ABB RAPID module: MAINMODULE

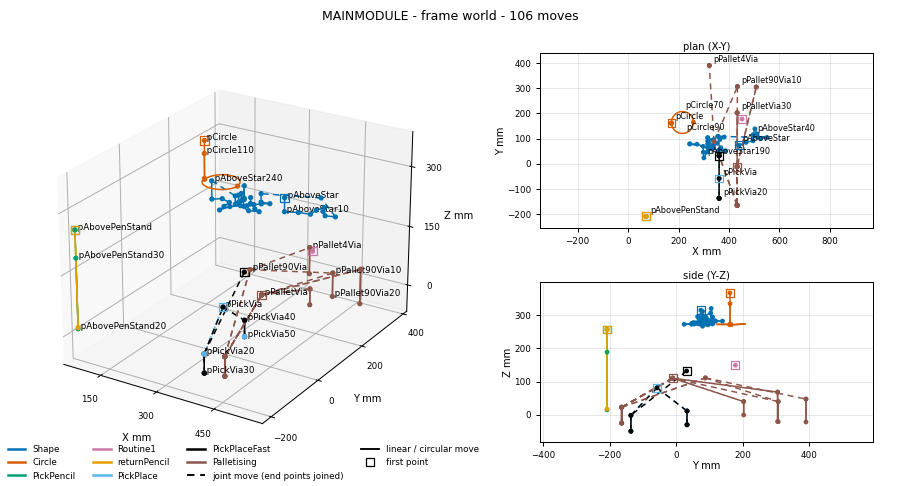
[picture p0: tool path of MAINMODULE in frame world, 106 of 141 moves have a stored position in this frame; points joined in program order, loops and branches not executed]
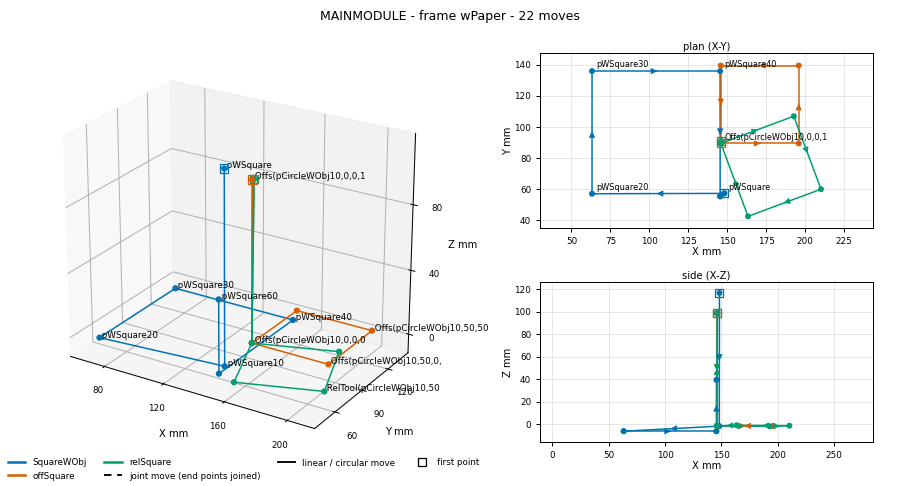
[picture p1: tool path of MAINMODULE in frame wPaper, 22 of 141 moves have a stored position in this frame; points joined in program order, loops and branches not executed]
MODULE MainModule
	CONST robtarget pAboveStar:=[[438.62,74.11,314.72],[0.00782336,-0.999705,-0.0203543,-0.0106794],[0,0,2,0],[9E+09,9E+09,9E+09,9E+09,9E+09,9E+09]];
	CONST robtarget pAboveStar10:=[[438.61,74.11,281.38],[0.00783533,-0.999705,-0.0203361,-0.0106734],[0,0,2,0],[9E+09,9E+09,9E+09,9E+09,9E+09,9E+09]];
	CONST robtarget pAboveStar20:=[[467.60,85.46,281.94],[0.00786178,-0.999706,-0.0202732,-0.0107677],[0,0,2,0],[9E+09,9E+09,9E+09,9E+09,9E+09,9E+09]];
	CONST robtarget pAboveStar30:=[[494.86,91.66,281.75],[0.00785369,-0.999704,-0.0202728,-0.010905],[0,0,2,0],[9E+09,9E+09,9E+09,9E+09,9E+09,9E+09]];
	CONST robtarget pAboveStar40:=[[495.39,115.61,282.55],[0.00784958,-0.999705,-0.0202499,-0.0109168],[0,0,2,0],[9E+09,9E+09,9E+09,9E+09,9E+09,9E+09]];
	CONST robtarget pAboveStar50:=[[502.60,139.11,282.02],[0.00780388,-0.999706,-0.0202427,-0.0108406],[0,0,2,0],[9E+09,9E+09,9E+09,9E+09,9E+09,9E+09]];
	CONST robtarget pAboveStar60:=[[511.39,118.70,282.17],[0.00782157,-0.999704,-0.0203071,-0.010834],[0,0,2,0],[9E+09,9E+09,9E+09,9E+09,9E+09,9E+09]];
	CONST robtarget pAboveStar70:=[[526.59,101.47,281.57],[0.00783068,-0.999704,-0.0203263,-0.0108239],[0,0,2,0],[9E+09,9E+09,9E+09,9E+09,9E+09,9E+09]];
	CONST robtarget pAboveStar80:=[[550.47,105.19,283.01],[0.00780734,-0.999704,-0.020355,-0.0107971],[0,0,2,0],[9E+09,9E+09,9E+09,9E+09,9E+09,9E+09]];
	CONST robtarget pAboveStar90:=[[513.27,105.19,320.11],[0.00778152,-0.999706,-0.0203135,-0.010705],[0,0,2,0],[9E+09,9E+09,9E+09,9E+09,9E+09,9E+09]];
	CONST robtarget pAboveStar100:=[[356.24,109.54,273.41],[0.0140382,0.0113166,0.999798,0.00891365],[0,0,0,0],[9E+09,9E+09,9E+09,9E+09,9E+09,9E+09]];
	CONST robtarget pAboveStar110:=[[381.12,106.70,276.14],[0.0141146,0.0112878,0.999797,0.00891807],[0,0,0,0],[9E+09,9E+09,9E+09,9E+09,9E+09,9E+09]];
	CONST robtarget pAboveStar120:=[[364.27,97.27,275.21],[0.0140659,0.0112485,0.999798,0.00892909],[0,0,0,0],[9E+09,9E+09,9E+09,9E+09,9E+09,9E+09]];
	CONST robtarget pAboveStar130:=[[353.90,82.53,276.31],[0.0142624,0.0112492,0.999794,0.00900628],[0,0,0,0],[9E+09,9E+09,9E+09,9E+09,9E+09,9E+09]];
	CONST robtarget pAboveStar140:=[[367.61,64.33,275.67],[0.0143661,0.0112371,0.999793,0.00904389],[0,0,0,0],[9E+09,9E+09,9E+09,9E+09,9E+09,9E+09]];
	CONST robtarget pAboveStar150:=[[386.45,52.10,277.62],[0.0144419,0.0112929,0.999791,0.00908413],[0,0,0,0],[9E+09,9E+09,9E+09,9E+09,9E+09,9E+09]];
	CONST robtarget pAboveStar160:=[[358.13,53.57,273.11],[0.0145648,0.011269,0.999789,0.00914371],[0,0,0,0],[9E+09,9E+09,9E+09,9E+09,9E+09,9E+09]];
	CONST robtarget pAboveStar170:=[[332.66,60.20,277.10],[0.0146625,0.0112876,0.999787,0.00917015],[0,0,0,0],[9E+09,9E+09,9E+09,9E+09,9E+09,9E+09]];
	CONST robtarget pAboveStar180:=[[313.01,46.92,275.35],[0.0146979,0.011265,0.999786,0.00921032],[0,0,0,0],[9E+09,9E+09,9E+09,9E+09,9E+09,9E+09]];
	CONST robtarget pAboveStar190:=[[300.34,23.93,272.39],[0.0147404,0.0112439,0.999785,0.00926598],[0,0,0,0],[9E+09,9E+09,9E+09,9E+09,9E+09,9E+09]];
	CONST robtarget pAboveStar200:=[[297.97,46.30,272.71],[0.0147271,0.0111926,0.999785,0.00933937],[0,0,0,0],[9E+09,9E+09,9E+09,9E+09,9E+09,9E+09]];
	CONST robtarget pAboveStar210:=[[297.39,69.49,273.85],[0.0147374,0.0111578,0.999785,0.00935574],[0,0,0,0],[9E+09,9E+09,9E+09,9E+09,9E+09,9E+09]];
	CONST robtarget pAboveStar220:=[[272.94,78.27,274.40],[0.0147777,0.0111411,0.999784,0.00940734],[0,0,0,0],[9E+09,9E+09,9E+09,9E+09,9E+09,9E+09]];
	CONST robtarget pAboveStar230:=[[244.38,79.32,266.59],[0.0148682,0.0111358,0.999783,0.00945356],[0,0,0,0],[9E+09,9E+09,9E+09,9E+09,9E+09,9E+09]];
	CONST robtarget pAboveStar240:=[[244.38,79.32,311.23],[0.0148422,0.0111395,0.999783,0.00942161],[0,0,0,0],[9E+09,9E+09,9E+09,9E+09,9E+09,9E+09]];
	CONST robtarget pAboveStar250:=[[356.24,109.54,293.90],[0.014005,0.0113197,0.999798,0.00888656],[0,0,0,0],[9E+09,9E+09,9E+09,9E+09,9E+09,9E+09]];
	CONST robtarget pAboveStar260:=[[316.18,64.48,295.54],[0.0148764,0.0111011,0.999783,0.00946381],[0,0,0,0],[9E+09,9E+09,9E+09,9E+09,9E+09,9E+09]];
	CONST robtarget pAboveStar270:=[[316.19,64.48,275.26],[0.0149083,0.0111043,0.999782,0.00947887],[0,0,0,0],[9E+09,9E+09,9E+09,9E+09,9E+09,9E+09]];
	CONST robtarget pAboveStar280:=[[319.92,71.32,275.46],[0.0149256,0.0110552,0.999782,0.00950374],[0,0,0,0],[9E+09,9E+09,9E+09,9E+09,9E+09,9E+09]];
	CONST robtarget pAboveStar290:=[[316.12,78.28,275.06],[0.0149297,0.0109983,0.999783,0.00948498],[0,0,0,0],[9E+09,9E+09,9E+09,9E+09,9E+09,9E+09]];
	CONST robtarget pAboveStar300:=[[316.12,78.28,292.53],[0.0149053,0.0110043,0.999784,0.00945692],[0,0,0,0],[9E+09,9E+09,9E+09,9E+09,9E+09,9E+09]];
	CONST robtarget pAboveStar310:=[[316.11,90.07,292.53],[0.0148157,0.0109983,0.999785,0.00941225],[0,0,0,0],[9E+09,9E+09,9E+09,9E+09,9E+09,9E+09]];
	CONST robtarget pAboveStar320:=[[316.13,90.08,275.06],[0.0150005,0.0109958,0.999782,0.00946723],[0,0,0,0],[9E+09,9E+09,9E+09,9E+09,9E+09,9E+09]];
	CONST robtarget pAboveStar330:=[[319.37,97.08,275.77],[0.015104,0.0109807,0.999781,0.009478],[0,0,0,0],[9E+09,9E+09,9E+09,9E+09,9E+09,9E+09]];
	CONST robtarget pAboveStar340:=[[315.40,103.87,275.53],[0.0151335,0.0110028,0.99978,0.00947056],[0,0,0,0],[9E+09,9E+09,9E+09,9E+09,9E+09,9E+09]];
	CONST robtarget pAboveStar350:=[[315.40,103.86,306.27],[0.0151151,0.0109962,0.999781,0.00943505],[0,0,0,0],[9E+09,9E+09,9E+09,9E+09,9E+09,9E+09]];
	CONST robtarget pAboveStar360:=[[335.06,68.19,290.35],[0.015148,0.0110168,0.99978,0.00946204],[0,0,0,0],[9E+09,9E+09,9E+09,9E+09,9E+09,9E+09]];
	CONST robtarget pAboveStar370:=[[336.39,68.12,273.72],[0.0152631,0.0109898,0.999778,0.0095098],[0,0,0,0],[9E+09,9E+09,9E+09,9E+09,9E+09,9E+09]];
	CONST robtarget pAboveStar380:=[[339.60,77.00,272.41],[0.0152849,0.0109759,0.999778,0.00952187],[0,0,0,0],[9E+09,9E+09,9E+09,9E+09,9E+09,9E+09]];
	CONST robtarget pAboveStar390:=[[341.03,87.53,273.01],[0.0152756,0.0109779,0.999778,0.0095199],[0,0,0,0],[9E+09,9E+09,9E+09,9E+09,9E+09,9E+09]];
	CONST robtarget pAboveStar400:=[[337.71,95.21,270.79],[0.015379,0.0110505,0.999775,0.00953919],[0,0,0,0],[9E+09,9E+09,9E+09,9E+09,9E+09,9E+09]];
	CONST robtarget pAboveStar410:=[[337.71,95.21,285.45],[0.0153497,0.0110536,0.999776,0.00950113],[0,0,0,0],[9E+09,9E+09,9E+09,9E+09,9E+09,9E+09]];
	CONST robtarget pCircle:=[[172.19,161.39,366.69],[0.0151956,0.0110729,0.999778,0.00948806],[0,-1,0,0],[9E+09,9E+09,9E+09,9E+09,9E+09,9E+09]];
	CONST robtarget pCircle10:=[[172.21,161.39,272.61],[0.0153553,0.0110984,0.999775,0.00956675],[0,-1,0,0],[9E+09,9E+09,9E+09,9E+09,9E+09,9E+09]];
	CONST robtarget pCircle30:=[[172.21,161.40,271.86],[0.0153361,0.0111049,0.999775,0.00957292],[0,-1,0,0],[9E+09,9E+09,9E+09,9E+09,9E+09,9E+09]];
	CONST robtarget pCircle20:=[[172.21,161.40,271.86],[0.0153361,0.0111049,0.999775,0.00957292],[0,-1,0,0],[9E+09,9E+09,9E+09,9E+09,9E+09,9E+09]];
	CONST robtarget pCircle40:=[[172.20,161.39,270.86],[0.0153246,0.0111176,0.999775,0.00958173],[0,-1,0,0],[9E+09,9E+09,9E+09,9E+09,9E+09,9E+09]];
	CONST robtarget pCircle60:=[[172.20,161.39,271.86],[0.0153102,0.0111183,0.999775,0.00956012],[0,-1,0,0],[9E+09,9E+09,9E+09,9E+09,9E+09,9E+09]];
	CONST robtarget pCircle50:=[[172.20,161.39,271.86],[0.0153102,0.0111183,0.999775,0.00956012],[0,-1,0,0],[9E+09,9E+09,9E+09,9E+09,9E+09,9E+09]];
	CONST robtarget pCircle80:=[[258.72,165.57,271.21],[0.0155733,0.0111395,0.999769,0.00972795],[0,-1,0,0],[9E+09,9E+09,9E+09,9E+09,9E+09,9E+09]];
	CONST robtarget pCircle70:=[[213.26,207.69,273.19],[0.0153849,0.0111178,0.999772,0.00975547],[0,-1,0,0],[9E+09,9E+09,9E+09,9E+09,9E+09,9E+09]];
	CONST robtarget pCircle100:=[[171.43,161.80,272.76],[0.0157088,0.0111,0.999768,0.00974234],[0,-1,0,0],[9E+09,9E+09,9E+09,9E+09,9E+09,9E+09]];
	CONST robtarget pCircle90:=[[217.30,120.93,272.13],[0.0155276,0.0111561,0.99977,0.00968626],[0,0,0,0],[9E+09,9E+09,9E+09,9E+09,9E+09,9E+09]];
	CONST robtarget pCircle110:=[[171.42,161.80,334.48],[0.0156731,0.0110978,0.999768,0.00974344],[0,-1,0,0],[9E+09,9E+09,9E+09,9E+09,9E+09,9E+09]];
	CONST robtarget pPen:=[[164.19,-206.82,447.81],[0.0140855,0.999796,-0.00773344,0.0122549],[-1,0,1,0],[9E+09,9E+09,9E+09,9E+09,9E+09,9E+09]];
	CONST robtarget pPen10:=[[164.19,-206.82,255.83],[0.014113,0.999795,-0.00772477,0.0122876],[-1,0,1,0],[9E+09,9E+09,9E+09,9E+09,9E+09,9E+09]];
	CONST robtarget pPen20:=[[164.19,-206.82,402.79],[0.0141017,0.999795,-0.00773661,0.0122669],[-1,0,1,0],[9E+09,9E+09,9E+09,9E+09,9E+09,9E+09]];
	CONST robtarget pWSquare:=[[148.16,57.39,116.56],[0.00760039,0.985996,-0.166519,0.00508158],[0,0,0,0],[9E+09,9E+09,9E+09,9E+09,9E+09,9E+09]];
	CONST robtarget pWSquare10:=[[148.04,57.38,-1.61],[0.00765696,0.985998,-0.166511,0.00489645],[0,0,0,0],[9E+09,9E+09,9E+09,9E+09,9E+09,9E+09]];
	CONST robtarget pWSquare20:=[[63.18,57.15,-6.08],[0.00767438,0.986016,-0.166404,0.00479981],[0,0,0,0],[9E+09,9E+09,9E+09,9E+09,9E+09,9E+09]];
	CONST robtarget pWSquare30:=[[63.20,135.93,-6.09],[0.00763878,0.986022,-0.166368,0.00484462],[0,0,0,0],[9E+09,9E+09,9E+09,9E+09,9E+09,9E+09]];
	CONST robtarget pWSquare40:=[[145.43,135.93,-6.09],[0.00764315,0.986027,-0.166343,0.00481764],[0,0,0,0],[9E+09,9E+09,9E+09,9E+09,9E+09,9E+09]];
	CONST robtarget pWSquare50:=[[145.46,55.49,-6.09],[0.00763597,0.986023,-0.166361,0.00488827],[0,0,0,0],[9E+09,9E+09,9E+09,9E+09,9E+09,9E+09]];
	CONST robtarget pWSquare60:=[[145.48,55.51,39.46],[0.00758059,0.986027,-0.16634,0.00490909],[0,0,0,0],[9E+09,9E+09,9E+09,9E+09,9E+09,9E+09]];
	CONST robtarget pAbovePenStand:=[[71.07,-207.77,256.82],[0.00907654,-0.0280649,0.999549,0.00556097],[-2,-1,-2,0],[9E+09,9E+09,9E+09,9E+09,9E+09,9E+09]];
	CONST robtarget pAbovePenStand10:=[[71.05,-207.81,17.76],[0.00903694,-0.0280484,0.999551,0.00548002],[-2,-1,-2,0],[9E+09,9E+09,9E+09,9E+09,9E+09,9E+09]];
	CONST robtarget pAbovePenStand20:=[[71.05,-207.84,14.94],[0.00903621,-0.0280371,0.999551,0.00543696],[-2,-1,-2,0],[9E+09,9E+09,9E+09,9E+09,9E+09,9E+09]];
	CONST robtarget pAbovePenStand30:=[[71.07,-207.82,188.80],[0.00907619,-0.0280604,0.99955,0.00546786],[-2,-1,-2,0],[9E+09,9E+09,9E+09,9E+09,9E+09,9E+09]];
	CONST robtarget pCircleWObj:=[[145.95,89.49,175.26],[0.00623942,0.984129,0.177325,-0.0027726],[-1,-1,-1,0],[9E+09,9E+09,9E+09,9E+09,9E+09,9E+09]];
	CONST robtarget pCircleWObj10:=[[145.91,89.49,-1.38],[0.00623623,0.984131,0.17731,-0.0028463],[-1,-1,-1,0],[9E+09,9E+09,9E+09,9E+09,9E+09,9E+09]];
	CONST robtarget pCircleWObj30:=[[59.69,88.08,-0.69],[0.00626669,0.984148,0.177212,-0.00309014],[-1,-1,-1,0],[9E+09,9E+09,9E+09,9E+09,9E+09,9E+09]];
	CONST robtarget pCircleWObj20:=[[104.28,44.81,0.78],[0.00625793,0.984143,0.17724,-0.00298966],[-1,-1,-1,0],[9E+09,9E+09,9E+09,9E+09,9E+09,9E+09]];
	CONST robtarget pCircleWObj50:=[[146.50,89.95,0.21],[0.00622075,0.984144,0.177231,-0.00332268],[-1,-1,-1,0],[9E+09,9E+09,9E+09,9E+09,9E+09,9E+09]];
	CONST robtarget pCircleWObj40:=[[102.61,131.54,-0.10],[0.00622868,0.984143,0.17724,-0.00320295],[-1,-1,-1,0],[9E+09,9E+09,9E+09,9E+09,9E+09,9E+09]];
	CONST robtarget pCircleWObj60:=[[146.53,89.93,120.78],[0.00626536,0.98414,0.17725,-0.00328061],[-1,-1,-1,0],[9E+09,9E+09,9E+09,9E+09,9E+09,9E+09]];
	CONST robtarget pTriangleWObj:=[[146.59,89.92,166.63],[0.00627944,0.984134,0.177285,-0.00319599],[-1,-1,-1,0],[9E+09,9E+09,9E+09,9E+09,9E+09,9E+09]];
	CONST robtarget pTriangleWObj10:=[[146.61,89.93,-1.46],[0.00627066,0.984138,0.177267,-0.00317229],[-1,-1,-1,0],[9E+09,9E+09,9E+09,9E+09,9E+09,9E+09]];
	CONST robtarget pTriangleWObj20:=[[72.70,56.70,-2.34],[0.00625777,0.984117,0.177377,-0.00333694],[-1,-1,-1,0],[9E+09,9E+09,9E+09,9E+09,9E+09,9E+09]];
	CONST robtarget pTriangleWObj30:=[[72.63,118.18,-0.40],[0.00623532,0.984124,0.177339,-0.00344523],[-1,-1,-1,0],[9E+09,9E+09,9E+09,9E+09,9E+09,9E+09]];
	CONST robtarget pTriangleWObj40:=[[146.62,89.92,123.42],[0.00628958,0.984135,0.17728,-0.00316079],[-1,-1,-1,0],[9E+09,9E+09,9E+09,9E+09,9E+09,9E+09]];
	CONST robtarget pPickVia:=[[360.73,-57.78,81.44],[0.00903673,-0.0280459,0.99955,0.00558822],[-1,-1,-1,0],[9E+09,9E+09,9E+09,9E+09,9E+09,9E+09]];
	CONST robtarget pPickVia10:=[[389.78,-126.91,12.64],[0.00911789,-0.0280836,0.999549,0.00553206],[-1,-1,-1,0],[9E+09,9E+09,9E+09,9E+09,9E+09,9E+09]];
	CONST robtarget pPickAbove10:=[[389.83,-126.95,-54.60],[0.00917495,-0.028089,0.999548,0.0054678],[-1,-1,-1,0],[9E+09,9E+09,9E+09,9E+09,9E+09,9E+09]];
	VAR clock cClock;
	VAR num nClock:=0;
	VAR string strClock:="";
	CONST robtarget pPickVia20:=[[360.72,-136.09,-1.19],[0.00903325,-0.0281173,0.999548,0.00555723],[-1,-1,-1,0],[9E+09,9E+09,9E+09,9E+09,9E+09,9E+09]];
	CONST robtarget pPickVia30:=[[360.77,-136.11,-48.89],[0.00910119,-0.0281037,0.999548,0.00552285],[-1,-1,-1,0],[9E+09,9E+09,9E+09,9E+09,9E+09,9E+09]];
	CONST robtarget pPickVia40:=[[360.83,32.61,11.70],[0.00906001,-0.0279562,0.999552,0.00563834],[0,0,0,0],[9E+09,9E+09,9E+09,9E+09,9E+09,9E+09]];
	CONST robtarget pPickVia50:=[[360.77,32.61,-29.56],[0.00898145,-0.0279684,0.999553,0.00563244],[0,0,0,0],[9E+09,9E+09,9E+09,9E+09,9E+09,9E+09]];
	CONST robtarget pPalletVia:=[[432.15,-10.57,110.48],[0.00897623,-0.0279392,0.999553,0.00565143],[-1,-1,-1,0],[9E+09,9E+09,9E+09,9E+09,9E+09,9E+09]];
	CONST robtarget pPalletVia10:=[[432.23,-163.79,23.13],[0.0089389,-0.0279646,0.999553,0.00565939],[-1,-1,-1,0],[9E+09,9E+09,9E+09,9E+09,9E+09,9E+09]];
	CONST robtarget pPalletVia20:=[[432.27,-163.81,-24.59],[0.00902617,-0.0279489,0.999553,0.00561107],[-1,-1,-1,0],[9E+09,9E+09,9E+09,9E+09,9E+09,9E+09]];
	CONST robtarget pPalletVia30:=[[432.16,202.87,40.09],[0.00885039,-0.0278895,0.999556,0.00567707],[0,0,0,0],[9E+09,9E+09,9E+09,9E+09,9E+09,9E+09]];
	CONST robtarget pPalletVia40:=[[432.15,202.88,-0.16],[0.00885213,-0.0278772,0.999556,0.00571044],[0,0,0,0],[9E+09,9E+09,9E+09,9E+09,9E+09,9E+09]];
	CONST robtarget pPallet90Via:=[[340.81,87.79,111.35],[0.00246793,-0.695514,0.7183,0.0172898],[-1,-1,-1,0],[9E+09,9E+09,9E+09,9E+09,9E+09,9E+09]];
	CONST robtarget pPallet90Via10:=[[433.23,306.73,40.16],[0.0024531,-0.695614,0.718204,0.0172648],[0,0,-1,0],[9E+09,9E+09,9E+09,9E+09,9E+09,9E+09]];
	CONST robtarget pPallet90Via20:=[[433.26,306.73,-20.32],[0.00247707,-0.6956,0.718218,0.0172488],[0,0,-1,0],[9E+09,9E+09,9E+09,9E+09,9E+09,9E+09]];
	CONST robtarget pPallet3Via:=[[507.97,304.84,68.59],[0.00881255,-0.0279233,0.999556,0.00560182],[0,0,0,0],[9E+09,9E+09,9E+09,9E+09,9E+09,9E+09]];
	CONST robtarget pPallet3Via10:=[[507.99,304.87,-19.58],[0.00883866,-0.0279657,0.999554,0.005633],[0,0,0,0],[9E+09,9E+09,9E+09,9E+09,9E+09,9E+09]];
	CONST robtarget pPallet4Via:=[[321.86,390.09,47.64],[0.00242,-0.695518,0.718297,0.0172813],[0,0,-1,0],[9E+09,9E+09,9E+09,9E+09,9E+09,9E+09]];
	CONST robtarget pPallet4Via10:=[[321.86,390.10,-21.25],[0.00243516,-0.695493,0.71832,0.0173165],[0,0,-1,0],[9E+09,9E+09,9E+09,9E+09,9E+09,9E+09]];
	PROC main()
		IF diSwitch1 = 1 AND diPenStand = 1 THEN
			PickPencil;
		ELSEIF diSwitch1 = 0 AND diPenStand = 0 THEN
			returnPencil;
		ENDIF
		IF diSwitch2 = 1 AND diGripSensor = 1 THEN
			nCircleNum := 0;
			FOR i FROM 1 TO 3 DO
				CircleWObj;
				Add nCircleNum, 1;
			ENDFOR
			UIMsgBox "3 circles drawn.";
		ELSEIF FALSE AND diGripSensor = 1 THEN
            nTriangleNum := 0;
			FOR i FROM 1 TO 3 DO
				TriangleWObj;
				Add nTriangleNum, 1;
			ENDFOR
			UIMsgBox "3 triangles drawn.";
		ELSEIF diSwitch4 = 1 THEN
			WHILE diSwitch4 = 1 DO
				Palletising;
			ENDWHILE
		ENDIF
	ENDPROC
	PROC Shape()
		MoveJ pAboveStar, v200, z20, tool0;
		MoveL pAboveStar10, v200, fine, tool0;
		MoveL pAboveStar20, v200, z50, tool0;
		MoveL pAboveStar30, v200, z0, tool0;
		MoveL pAboveStar40, v200, z50, tool0;
		MoveL pAboveStar50, v200, z0, tool0;
		MoveL pAboveStar60, v200, z50, tool0;
		MoveL pAboveStar70, v200, z0, tool0;
		MoveL pAboveStar80, v200, fine, tool0;
		MoveJ pAboveStar90, v200, fine, tool0;
		MoveJ pAboveStar250, v200, fine, tool0;
		MoveL pAboveStar100, v200, z50, tool0;
		MoveL pAboveStar110, v200, z0, tool0;
		MoveL pAboveStar120, v200, z50, tool0;
		MoveL pAboveStar130, v200, z0, tool0;
		MoveL pAboveStar140, v200, z50, tool0;
		MoveL pAboveStar150, v200, z0, tool0;
		MoveL pAboveStar160, v200, z50, tool0;
		MoveL pAboveStar170, v200, z0, tool0;
		MoveL pAboveStar180, v200, z50, tool0;
		MoveL pAboveStar190, v200, z0, tool0;
		MoveL pAboveStar200, v200, z50, tool0;
		MoveL pAboveStar210, v200, z0, tool0;
		MoveL pAboveStar220, v200, z50, tool0;
		MoveL pAboveStar230, v200, z0, tool0;
		MoveL pAboveStar240, v200, fine, tool0;
		MoveJ pAboveStar260, v200, fine, tool0;
		MoveL pAboveStar270, v200, z0, tool0;
		MoveL pAboveStar280, v200, z50, tool0;
		MoveL pAboveStar290, v200, z0, tool0;
		MoveL pAboveStar300, v200, fine, tool0;
		MoveJ pAboveStar310, v200, fine, tool0;
		MoveL pAboveStar320, v200, z0, tool0;
		MoveL pAboveStar330, v200, z50, tool0;
		MoveL pAboveStar340, v200, z50, tool0;
		MoveL pAboveStar350, v200, z50, tool0;
		MoveL pAboveStar360, v200, fine, tool0;
		MoveL pAboveStar370, v200, z0, tool0;
		MoveL pAboveStar380, v200, z50, tool0;
		MoveL pAboveStar390, v200, z50, tool0;
		MoveL pAboveStar400, v200, z0, tool0;
		MoveL pAboveStar410, v200, fine, tool0;
	ENDPROC
	PROC Circle()
		MoveJ pCircle, v1000, z50, tool0;
		MoveL pCircle40, v1000, z50, tool0;
		MoveC pCircle70, pCircle80, v200, fine, tool0;
		MoveC pCircle90, pCircle100, v200, fine, tool0;
		MoveL pCircle110, v200, z50, tool0;
	ENDPROC
	PROC PickPencil()
		Set doGripper;
		MoveJ pAbovePenStand, v100, fine, toolPencil;
		MoveL pAbovePenStand20, v40, fine, toolPencil;
		Reset doGripper;
		WaitTime 0.5;
		MoveL pAbovePenStand30, v40, fine, toolPencil;
	ENDPROC
	PROC Routine1()
		MoveL [[451.82,177.96,149.37],[0.0180374,-0.0179567,0.999633,-0.0092314],[0,-1,0,0],[9E+09,9E+09,9E+09,9E+09,9E+09,9E+09]], v1000, z50, toolPencil;
	ENDPROC
	PROC SquareWObj()
		MoveJ pWSquare, v200, z20, toolPencil\WObj:=wPaper;
		MoveL pWSquare10, v40, fine, toolPencil\WObj:=wPaper;
		MoveL pWSquare20, v40, fine, toolPencil\WObj:=wPaper;
		MoveL pWSquare30, v40, fine, toolPencil\WObj:=wPaper;
		MoveL pWSquare40, v40, fine, toolPencil\WObj:=wPaper;
		MoveL pWSquare50, v40, fine, toolPencil\WObj:=wPaper;
		MoveL pWSquare60, v40, fine, toolPencil\WObj:=wPaper;
	ENDPROC
	PROC Triangle()
		<SMT>
	ENDPROC
	PROC returnPencil()
		MoveJ pAbovePenStand, v100, fine, toolPencil;
		MoveL pAbovePenStand10, v40, fine, toolPencil;
		Set doGripper;
		WaitTime 0.5;
		MoveL pAbovePenStand, v40, fine, toolPencil;
	ENDPROC
	PROC returnHome()
		MoveJ pHome, v100, fine, toolPencil;
	ENDPROC
	PROC CircleWObj()
		!MoveJ pCircleWObj, v100, fine, toolPencil\WObj:=wPaper;
		!MoveL pCircleWObj10, v100, fine, toolPencil\WObj:=wPaper;
		!MoveC pCircleWObj20, pCircleWObj30, v100, fine, toolPencil\WObj:=wPaper;
		!MoveC pCircleWObj40, pCircleWObj50, v100, fine, toolPencil\WObj:=wPaper;
		!MoveL pCircleWObj60, v100, fine, toolPencil\WObj:=wPaper;
        MoveJ Offs(pCircleWObj,10*nCircleNum,0,0), v100, fine, toolPencil\WObj:=wPaper;
		MoveL Offs(pCircleWObj10,10*nCircleNum,0,0), v100, fine, toolPencil\WObj:=wPaper;
		MoveC Offs(pCircleWObj20,10*nCircleNum,0,0), Offs(pCircleWObj30,10*nCircleNum,0,0), v100, fine, toolPencil\WObj:=wPaper;
		MoveC Offs(pCircleWObj40,10*nCircleNum,0,0), Offs(pCircleWObj50,10*nCircleNum,0,0), v100, fine, toolPencil\WObj:=wPaper;
		MoveL Offs(pCircleWObj60,10*nCircleNum,0,0), v100, fine, toolPencil\WObj:=wPaper;
	ENDPROC
	PROC TriangleWObj()
		MoveJ Offs(pTriangleWObj,10*nTriangleNum,0,0), v100, fine, toolPencil\WObj:=wPaper;
		MoveL Offs(pTriangleWObj10,10*nTriangleNum,0,0), v40, fine, toolPencil\WObj:=wPaper;
		MoveL Offs(pTriangleWObj20,10*nTriangleNum,0,0), v40, fine, toolPencil\WObj:=wPaper;
		MoveL Offs(pTriangleWObj30,10*nTriangleNum,0,0), v40, fine, toolPencil\WObj:=wPaper;
		MoveL Offs(pTriangleWObj10,10*nTriangleNum,0,0), v40, fine, toolPencil\WObj:=wPaper;
		MoveL Offs(pTriangleWObj40,10*nTriangleNum,0,0), v100, fine, toolPencil\WObj:=wPaper;
	ENDPROC
	PROC PrintExercise()
		nMyNum := 9;
		IF nMyNum < 5 THEN
			TPWrite "My number is lower than 5 ";
		ELSEIF nMyNum < 10 THEN
			TPWrite "My number is lower than 10 ";
		ELSE
			TPWrite "My number is:"\Num:=nMyNum;
		ENDIF
	ENDPROC
	PROC offSquare()
		ClkReset cClock;
		ClkStart cClock;
		MoveJ Offs(pCircleWObj10,0,0,100), v100, fine, toolPencil\WObj:=wPaper;
		MoveL Offs(pCircleWObj10,0,0,0), v100, fine, toolPencil\WObj:=wPaper;
		MoveL Offs(pCircleWObj10,50,0,0), v100, fine, toolPencil\WObj:=wPaper;
		MoveL Offs(pCircleWObj10,50,50,0), v100, fine, toolPencil\WObj:=wPaper;
		MoveL Offs(pCircleWObj10,0,50,0), v100, fine, toolPencil\WObj:=wPaper;
		MoveL Offs(pCircleWObj10,0,0,0), v100, fine, toolPencil\WObj:=wPaper;
		MoveL Offs(pCircleWObj10,0,0,100), v100, fine, toolPencil\WObj:=wPaper;
		ClkStop clock1;
		nClock := ClkRead(cClock);
		strClock := ValToStr(nClock);
		UIMsgBox strClock;
	ENDPROC
	PROC relSquare()
		MoveJ RelTool(pCircleWObj10,0,0,-100), v100, fine, toolPencil\WObj:=wPaper;
		MoveJ RelTool(pCircleWObj10,0,0,-100\Rx:=30\Rz:=30), v100, fine, toolPencil\WObj:=wPaper;
		MoveL RelTool(pCircleWObj10,0,0,0\Rx:=30\Rz:=30), v100, fine, toolPencil\WObj:=wPaper;
		MoveL RelTool(pCircleWObj10,50,0,0\Rx:=30\Rz:=30), v100, fine, toolPencil\WObj:=wPaper;
		MoveL RelTool(pCircleWObj10,50,50,0\Rx:=30\Rz:=30), v100, fine, toolPencil\WObj:=wPaper;
		MoveL RelTool(pCircleWObj10,0,50,0\Rx:=30\Rz:=30), v100, fine, toolPencil\WObj:=wPaper;
		MoveL RelTool(pCircleWObj10,0,0,0\Rx:=30\Rz:=30), v100, fine, toolPencil\WObj:=wPaper;
		MoveL RelTool(pCircleWObj10,0,0,-100), v100, fine, toolPencil\WObj:=wPaper;
	ENDPROC
	PROC PickPlace()
		ClkReset cClock;
		ClkStart cClock;
		Set doGripper;
		MoveJ pPickVia, v100, z50, toolPencil;
		MoveJ pPickVia20, v100, z50, toolPencil;
		MoveL pPickVia30, v100, fine, toolPencil;
		Reset doGripper;
		Set doMagnet;
		WaitTime 1;
		MoveL pPickVia30, v100, z50, toolPencil;
		MoveJ pPickVia20, v100, z50, toolPencil;
		MoveJ pPickVia, v100, z50, toolPencil;
		MoveJ pPickVia40, v100, z50, toolPencil;
		MoveL pPickVia50, v100, fine, toolPencil;
		Set doGripper;
		Reset doMagnet;
		WaitTime 1;
		MoveL pPickVia50, v100, fine, toolPencil;
		MoveJ pPickVia40, v100, z50, toolPencil;
		ClkStop cClock;
		TPWrite "Cycle time: "\Num:=ClkRead(cClock);
	ENDPROC
	PROC PickPlaceFast()
		ClkReset cClock;
		ClkStart cClock;
		Set doGripper;
		MoveJ [[360.73,31.38,132.06],[0.0090413,-0.0279876,0.999552,0.00561662],[0,0,0,0],[9E+09,9E+09,9E+09,9E+09,9E+09,9E+09]], v100, z50, toolPencil;
		MoveJ pPickVia20, v100, z50, toolPencil;
		MoveL pPickVia30, v100, fine, toolPencil;
		Reset doGripper;
		Set doMagnet;
		WaitTime 1;
		MoveL pPickVia30, v100, z50, toolPencil;
		MoveJ pPickVia20, v100, z50, toolPencil;
		MoveJ pPickVia, v100, z50, toolPencil;
		MoveJ pPickVia40, v100, z50, toolPencil;
		MoveL pPickVia50, v100, fine, toolPencil;
		Set doGripper;
		Reset doMagnet;
		WaitTime 1;
		MoveL pPickVia50, v100, fine, toolPencil;
		MoveJ pPickVia40, v100, z50, toolPencil;
		ClkStop cClock;
		TPWrite "Cycle time: "\Num:=ClkRead(cClock);
	ENDPROC
	PROC RevCounter()
		MoveAbsJ [[0,0,0,0,0,0],[9E+09,9E+09,9E+09,9E+09,9E+09,9E+09]]\NoEOffs, v100, z50, toolPencil;
	ENDPROC
	PROC Palletising()
		MoveJ pPalletVia, v1000, z200, toolPencil;
		WaitDI diSwitch3, 0;
		MoveJ pPalletVia10, v1000, z200, toolPencil;
		MoveL pPalletVia20, v1000, fine, toolPencil;
		Set doMagnet;
		WaitTime 0.25;
		MoveL pPalletVia10, v1000, z200, toolPencil;
		MoveJ pPalletVia, v1000, z200, toolPencil;
		MoveJ pPalletVia30, v1000, z200, toolPencil;
		MoveL pPalletVia40, v1000, fine, toolPencil;
		Reset doMagnet;
		WaitTime 0.25;
		MoveL pPalletVia30, v1000, z50, toolPencil;
		!2
		MoveJ pPalletVia, v1000, z200, toolPencil;
		WaitDI diSwitch3, 1;
		MoveJ pPalletVia10, v1000, z200, toolPencil;
		MoveL pPalletVia20, v1000, fine, toolPencil;
		Set doMagnet;
		WaitTime 0.25;
		MoveL pPalletVia10, v1000, z200, toolPencil;
		MoveJ pPallet90Via, v1000, z200, toolPencil;
		MoveJ pPallet90Via10, v1000, z200, toolPencil;
		MoveL pPallet90Via20, v1000, fine, toolPencil;
		Reset doMagnet;
		WaitTime 0.25;
		MoveL pPallet90Via10, v1000, z200, toolPencil;
		!3
		MoveJ pPalletVia, v1000, z200, toolPencil;
		WaitDI diSwitch3, 0;
        MoveJ pPalletVia10, v1000, z200, toolPencil;
		MoveL pPalletVia20, v1000, fine, toolPencil;
		Set doMagnet;
		WaitTime 0.25;
		MoveL pPalletVia10, v1000, z200, toolPencil;
		MoveJ pPalletVia, v1000, z200, toolPencil;
		MoveJ pPallet3Via, v1000, z200, toolPencil;
		MoveL pPallet3Via10, v1000, fine, toolPencil;
		Reset doMagnet;
		WaitTime 0.25;
		MoveL pPallet3Via, v1000, z50, toolPencil;
        !4
        MoveJ pPalletVia, v1000, z200, toolPencil;
		WaitDI diSwitch3, 1;
		MoveJ pPalletVia10, v1000, z200, toolPencil;
		MoveL pPalletVia20, v1000, fine, toolPencil;
		Set doMagnet;
		WaitTime 0.25;
		MoveL pPalletVia10, v1000, z200, toolPencil;
		MoveJ pPallet90Via, v1000, z200, toolPencil;
		MoveJ pPallet4Via, v1000, z200, toolPencil;
		MoveL pPallet4Via10, v1000, fine, toolPencil;
		Reset doMagnet;
		WaitTime 0.25;
		MoveL pPallet4Via, v1000, z200, toolPencil;
	ENDPROC
ENDMODULE
